FUNCTION Convert_DATE_TO_SINT : Hresult
VAR_INPUT
	in : DATE;
	out : REFERENCE TO SINT;
END_VAR
VAR
	converted : SINT;
END_VAR

converted := DATE_TO_SINT(in);

IF (SINT_TO_DATE(converted) <> in) THEN
	Convert_DATE_TO_SINT := INCOMPATIBLE;
	RETURN;
END_IF

out := converted;

END_FUNCTION

(* stored: Version 1.1.0.1, ProductVersion 3.1.4024.12
   POU Convert_DATE_TO_SINT: Id {023183cb-bd59-44f5-a338-855946189d7d}, SpecialFunc None *)
